Staubli VAL3: onProgEnd.pgx

public program onProgEnd(string& x_sItem[])
begin
end
